Fanuc KAREL source: CNV_STR_CONF.kl

PROGRAM T
%NOLOCKGROUP
VAR
 v0 : STRING[40]
 v1 : CONFIG
 v2 : INTEGER
BEGIN
 CNV_STR_CONF(v0, v1, v2)
END T
